(* Provides basic string builder implementation.
IMPORTANT NOTE! Doing too many method chains might cause the codesys compiler to either be very slow
when doing the "generating code" part or even fail. Restrain to not using too many or too
many nested methods ( method(fb.Method(fb2.Method())... ).
*)
FUNCTION_BLOCK FB_StringBuilderBase IMPLEMENTS I_StringBuilderBase
VAR
	_string	: Tc2_System.T_MaxString;
END_VAR

(* Adds a string to the build sequence.*)
METHOD AddString : I_StringBuilderBase
VAR_INPUT
	(* String to be added.*)
	str	: Tc2_System.T_MaxString;
END_VAR
_string := Tc2_Standard.CONCAT(
	STR1 := _string, 
	STR2 := str);
	
AddString := THIS^;
END_METHOD

(* Adds a string to the build sequence and wraps the str in double quotation marks "str"*)
METHOD AddWithDblQuotationMarks : I_StringBuilderBase
VAR_INPUT
	str	: Tc2_System.T_MaxString;
END_VAR
_string := Tc2_Standard.CONCAT(
	STR1 := _string, 
	STR2 := Tc2_Standard.CONCAT(
		STR1 := StringConstants.DoubleQuotationMark, 
		STR2 := Tc2_Standard.CONCAT(
			STR1 := str, 
			STR2 := StringConstants.DoubleQuotationMark))); 
	
AddWithDblQuotationMarks := THIS^;
END_METHOD

(* Adds a string to the build sequence and wraps the str in quotation marks 'str'*)
METHOD AddWithQuotationMark : I_StringBuilderBase
VAR_INPUT
	str	: Tc2_System.T_MaxString;
END_VAR
_string := Tc2_Standard.CONCAT(
	STR1 := _string, 
	STR2 := Tc2_Standard.CONCAT(
		STR1 := StringConstants.SingleQuotationMark, 
		STR2 := Tc2_Standard.CONCAT(
			STR1 := str, 
			STR2 := StringConstants.SingleQuotationMark))); 
		
AddWithQuotationMark := THIS^;
END_METHOD

(* Finishes string generation and returns the generated string*)
METHOD Create : Tc2_System.T_MaxString
Create := _string;
END_METHOD

(* Reset the string build sequence, clear any string built so far.*)
METHOD Reset : I_StringBuilderBase
_string := '';
Reset := THIS^;
END_METHOD

END_FUNCTION_BLOCK

(* stored: Version 1.1.0.1, ProductVersion 3.1.4024.14
   POU FB_StringBuilderBase: Id {4af2ae7b-34e5-0402-2ab5-b787ed381493}, SpecialFunc None
   Method AddString: Id {a1f2665a-9e23-0057-3cb2-001019efbfb5}
   Method AddWithDblQuotationMarks: Id {0e9fd4de-15c4-07a9-0872-3820188174d7}
   Method AddWithQuotationMark: Id {71b839a6-f4de-0e1d-0723-bae3b89369d5}
   Method Create: Id {837ad951-dde3-0ecc-1e91-80edffc6563f}
   Method Reset: Id {c0b64bb0-ab5a-04e6-313f-3575f6a54110} *)
